{attribute 'qualified_only'}
{attribute 'strict'}
TYPE GuidanceSystemSTM :
(
	Idling,
	Initialising,
	PreRunning,
	Running,
	PostRunning
);
END_TYPE

(* stored: Version 1.1.0.1, ProductVersion 3.1.4024.12
   DUT GuidanceSystemSTM: Id {4f1c65d1-df72-4db4-9416-57d142abfa9e} *)
